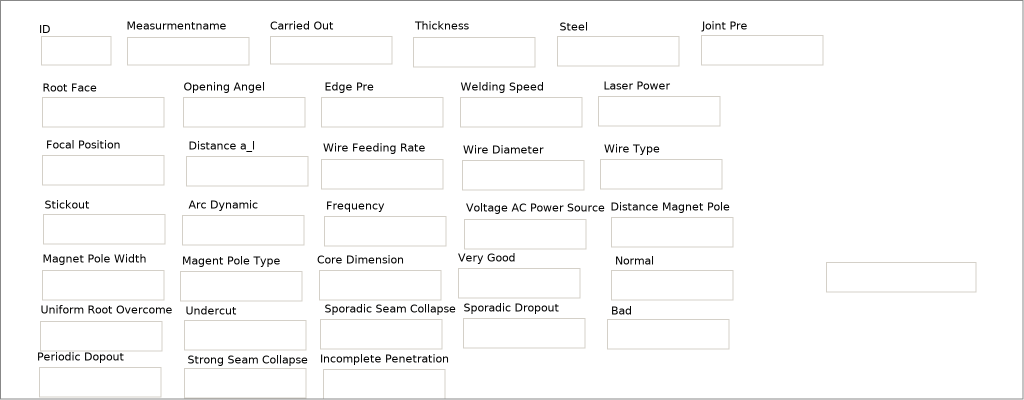
VISUALIZATION Write_Metadata_Visu  // 1024x400
    Textfield (41,36 70x29), text variable: GVL_Meta.Id
        OnMouseDown: write the text variable via Default
    Label (10,15 70x29), "ID"
    Group (117,13 132x52), text variable: GVL_Meta.measurementname
        Textfield (10,24 122x28), text variable: GVL_Meta.Id
        Label (0,0 119x26), "Measurmentname"
    Group (264,13 128x55), text variable: GVL_Meta.carried_out
        Textfield (6,23 122x28), text variable: GVL_Meta.Id
        Label (0,0 76x26), "Carried Out"
    Group (404,12 131x55), text variable: GVL_Meta.thickness
        Textfield (9,25 122x30), text variable: GVL_Meta.Id
        Label (0,0 76x28), "Thickness"
    Group (545,13 134x53), text variable: GVL_Meta.steel
        Textfield (12,23 122x30), text variable: GVL_Meta.Id
        Label (0,0 58x28), "Steel"
    Group (696,12 127x53), text variable: GVL_Meta.joint_pre
        Textfield (5,23 122x30), text variable: GVL_Meta.Id
        Label (0,0 58x28), "Joint Pre"
    Group (41,74 123x53), text variable: GVL_Meta.root_face
        Textfield (1,23 122x30), text variable: GVL_Meta.Id
        Label (0,0 58x28), "Root Face"
    Group (167,73 138x54), text variable: GVL_Meta.opening_angel
        Textfield (16,24 122x30), text variable: GVL_Meta.Id
        Label (0,0 115x28), "Opening Angel"
    Group (316,73 127x54), text variable: GVL_Meta.edge_pre
        Textfield (5,24 122x30), text variable: GVL_Meta.Id
        Label (0,0 67x28), "Edge Pre"
    Group (451,73 131x54), text variable: GVL_Meta.welding_speed
        Textfield (9,24 122x30), text variable: GVL_Meta.Id
        Label (0,0 103x28), "Welding Speed"
    Group (588,72 132x54), text variable: GVL_Meta.laser_power
        Textfield (10,24 122x30), text variable: GVL_Meta.Id
        Label (0,0 98x28), "Laser Power"
    Group (26,131 138x54), text variable: GVL_Meta.focal_position
        Textfield (16,24 122x30), text variable: GVL_Meta.Id
        Label (0,0 115x28), "Focal Position"
    Group (173,132 135x54), text variable: GVL_Meta.distance_a_l
        Textfield (13,24 122x30), text variable: GVL_Meta.Id
        Label (0,0 98x28), "Distance a_l"
    Group (317,134 126x55), text variable: GVL_Meta.wire_feeding_rate
        Textfield (4,25 122x30), text variable: GVL_Meta.Id
        Label (0,0 115x28), "Wire Feeding Rate"
    Group (446,136 138x54), text variable: GVL_Meta.wire_diameter
        Textfield (16,24 122x30), text variable: GVL_Meta.Id
        Label (0,0 115x28), "Wire Diameter"
    Group (589,135 133x54), text variable: GVL_Meta.wire_type
        Textfield (11,24 122x30), text variable: GVL_Meta.Id
        Label (0,0 86x28), "Wire Type"
    Group (33,191 132x53), text variable: GVL_Meta.stickout
        Textfield (10,23 122x30), text variable: GVL_Meta.Id
        Label (0,0 68x28), "Stickout"
    Group (166,191 138x54), text variable: GVL_Meta.arc_dynamic
        Textfield (16,24 122x30), text variable: GVL_Meta.Id
        Label (0,0 115x28), "Arc Dynamic"
    Group (298,192 148x54), text variable: GVL_Meta.frequency
        Textfield (26,24 122x30), text variable: GVL_Meta.Id
        Label (0,0 115x28), "Frequency"
    Group (454,194 163x55), text variable: GVL_Meta.voltage_ac_power_source
        Textfield (10,25 122x30), text variable: GVL_Meta.Id
        Label (0,0 163x28), "Voltage AC Power Source"
    Group (603,193 135x54), text variable: GVL_Meta.distance_magnet_pole
        Textfield (8,24 122x30), text variable: GVL_Meta.Id
        Label (0,0 135x28), "Distance Magnet Pole"
    Group (37,245 127x55), text variable: GVL_Meta.magnet_pole_width
        Textfield (5,25 122x30), text variable: GVL_Meta.Id
        Label (0,0 115x28), "Magnet Pole Width"
    Group (174,247 128x54), text variable: GVL_Meta.magnet_pole_type
        Textfield (6,24 122x30), text variable: GVL_Meta.Id
        Label (0,0 115x28), "Magent Pole Type"
    Group (303,246 138x54), text variable: GVL_Meta.core_dimension
        Textfield (16,24 122x30), text variable: GVL_Meta.Id
        Label (0,0 115x28), "Core Dimension"
    Group (440,244 140x54), text variable: GVL_Meta.very_good
        Textfield (18,24 122x30), text variable: GVL_Meta.Id
        Label (0,0 94x28), "Very Good"
    Group (601,247 132x53), text variable: GVL_Meta.normal
        Textfield (10,23 122x30), text variable: GVL_Meta.Id
        Label (0,0 67x28), "Normal"
    Group (32,296 149x55), text variable: GVL_Meta.uniform_root_overcome
        Textfield (8,25 122x30), text variable: GVL_Meta.Id
        Label (0,0 149x28), "Uniform Root Overcome"
    Group (172,297 134x53), text variable: GVL_Meta.undercut
        Textfield (12,23 122x30), text variable: GVL_Meta.Id
        Label (0,0 78x28), "Undercut"
    Group (315,295 151x54), text variable: GVL_Meta.sporadic_seam_collapse
        Textfield (5,24 122x30), text variable: GVL_Meta.Id
        Label (0,0 151x28), "Sporadic Seam Collapse"
    Group (454,294 131x54), text variable: GVL_Meta.sporadic_dropout
        Textfield (9,24 122x30), text variable: GVL_Meta.Id
        Label (0,0 115x28), "Sporadic Dropout"
    Group (589,297 140x52), text variable: GVL_Meta.bad
        Textfield (18,22 122x30), text variable: GVL_Meta.Id
        Label (0,0 65x28), "Bad"
    Group (23,343 138x54), text variable: GVL_Meta.periodic_dropout
        Textfield (16,24 122x30), text variable: GVL_Meta.Id
        Label (0,0 115x28), "Periodic Dopout"
    Group (180,346 136x52), text variable: GVL_Meta.strong_seam_collapse
        Textfield (4,22 122x30), text variable: GVL_Meta.Id
        Label (0,0 136x28), "Strong Seam Collapse"
    Group (307,345 155x54), text variable: GVL_Meta.incomplite_penetration
        Textfield (16,24 122x30), text variable: GVL_Meta.Id
        Label (0,0 155x28), "Incomplete Penetration"
    Textfield (826,262 150x30)
END_VISUALIZATION

(* stored: Version 1.1.0.1, ProductVersion 3.1.4024.12
   Visu Write_Metadata_Visu: Id {91455096-e802-472c-aee2-3d13801c3992} *)
